// TIA Portal V20 export
// export: Created 2025-12-01T14:56:12.1884079Z, ExportSetting None, DisplayName Totally Integrated Automation Portal, DisplayVersion V20 Update 3, DisplayName TIA Portal Openness, DisplayVersion V20 Update 3, DisplayName TIA Portal Version Control Interface, DisplayVersion V20 Update 3, DisplayName STEP 7 Professional, DisplayVersion V20 Update 3, DisplayName STEP 7 Safety, DisplayVersion V20 Update 2, DisplayName WinCC Basic/Comfort/Advanced, DisplayVersion V20 Update 3, DisplayName WinCC Professional, DisplayVersion V20 Update 3, DisplayName WinCC Unified, DisplayVersion V20 Update 3
TYPE "Selector"
   STRUCT
      U8 : Bool;
      U9 : Bool;
      Libre_02 : Bool;
      Libre_03 : Bool;
      Libre_04 : Bool;
      Libre_05 : Bool;
      Libre_06 : Bool;
      Libre_07 : Bool;
      U0 : Bool;
      U1 : Bool;
      U2 : Bool;
      U3 : Bool;
      U4 : Bool;
      U5 : Bool;
      U6 : Bool;
      U7 : Bool;
   END_STRUCT;
END_TYPE
